{attribute 'GeneratedUsingTerminal: EK1122-0000-0018'}
{attribute addProperty BoxType "EK1122-0000-0018"}
{attribute addProperty Id "Beckhoff_EL33xxsub_EK1100EK1100_AB5A94672"}
{attribute addProperty CRC "494744280"}
{attribute addProperty Size "2"}
TYPE Beckhoff_EL33xxEK1122_1D7D32D8 EXTENDS EK1122_AB5A9467 :
STRUCT
	{attribute addProperty Name "Beckhoff_EL33xxsub_EK1100"}
	Beckhoff_EL33xxsub_EK1100 : EK1100_AB5A9467;
END_STRUCT
END_TYPE

(* stored: Version 1.2.0.0, ProductVersion 3.1.4024.9
   DUT Beckhoff_EL33xxEK1122_1D7D32D8: Id {ae0f1f46-0e53-4da6-95db-8315739ae6b6} *)
